Universal Robots PolyScope program: usb.urp

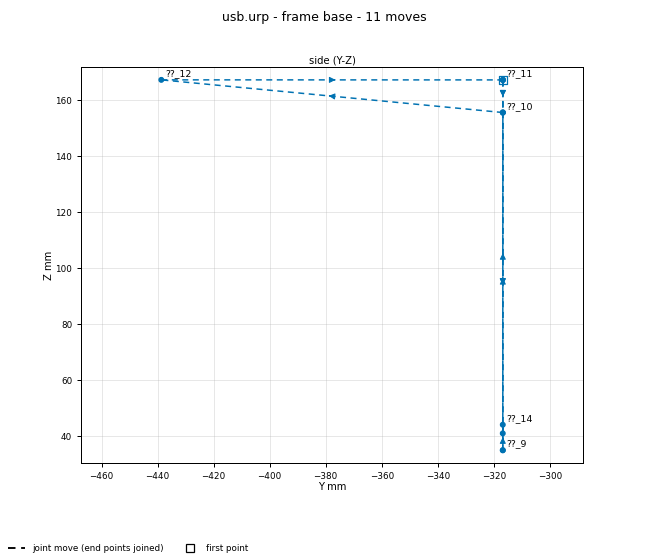
[picture p0: tool path of usb.urp in frame base, 11 of 11 moves have a stored position in this frame; points joined in program order, loops and branches not executed]
Program usb (installation=20240827 directory=/programs createdIn=5.15.1 lastSavedIn=5.15.1 robotSerialNumber=20245500285)
Calibrated DH parameters: a=[0.000097, -0.210459, -0.026602, 0.000137, 0.000078, 0]; d=[0.162601, 254.180657, -54.076236, -199.970743, 0.099615, 0.099684]; alpha=[1.569796, -0.001455, 0.001957, 1.570525, -1.571561, 0]; deltaTheta=[0, -1.053331, 8.839472, -1.50296, 0.000002, 0]
InitVariablesNode
Robot Program (runOnlyOnce=false)
  Script: usb = rpc_factory("xmlrpc","http://192.168.1.7:9120/RPC2")
  SuppressedNode
    MoveJ speed 60 deg/s, acceleration 80 deg/s^2 (useActiveTCP=true) feature=Base
      SuppressedNode
        Waypoint 路点_1: TCP in base x=280.909 y=-438.416 z=138.453 mm, rx=-0.0039 ry=2.6174 rz=0.002 rad; joints [90, -89.997, 120, -119.999, -60.002, 0] deg; TCP offset x=-0.17 y=0 z=192.95 mm, rx=0 ry=0 rz=0 rad
      Popup Message (haltProgram=false message=1 inputType=Text)
      Waypoint 路点_7: TCP in base x=280.9 y=-438.411 z=138.447 mm, rx=-0.0038 ry=3.1416 rz=0 rad; joints [107.671, -84.178, 107.406, -113.272, -90.026, 17.702] deg
      Waypoint 路点_2: TCP in base x=300.223 y=-316.781 z=157.956 mm, rx=0.0118 ry=-3.1414 rz=0.0001 rad; joints [115.532, -97.131, 117.117, -110.029, -90.021, 25.257] deg
      Waypoint 路点_3: TCP in base x=300.251 y=-316.773 z=100.612 mm, rx=0.0108 ry=-2.8383 rz=-0.0015 rad; joints [125.162, -84.56, 113.268, -108.499, -104.146, 36.158] deg
      Waypoint 路点_4: TCP in base x=300.243 y=-316.792 z=44.753 mm, rx=0.0106 ry=-2.8383 rz=-0.0015 rad; joints [125.158, -79.995, 117.672, -117.469, -104.165, 36.163] deg
      SuppressedNode
        Waypoint 路点_5: TCP in base x=301.229 y=-316.057 z=44.799 mm, rx=-0.0007 ry=-3.106 rz=-0.1207 rad; joints [115.546, -85.69, 123.783, -123.302, -89.838, 25.723] deg
      SuppressedNode
        Waypoint 路点_6: TCP in base x=280.91 y=-438.41 z=138.456 mm, rx=-0.0038 ry=2.6174 rz=0.002 rad; joints [89.999, -89.998, 120.001, -119.999, -60.001, 0.001] deg
      Waypoint ccc: TCP in base x=300.236 y=-316.791 z=40.853 mm, rx=0.0106 ry=-2.8383 rz=-0.0015 rad; joints [125.157, -79.629, 117.939, -118.1, -104.166, 36.162] deg
      Popup Message (haltProgram=false message=2 inputType=Text)
      Waypoint bbb: TCP in base x=300.214 y=-316.776 z=46.329 mm, rx=0.0105 ry=-3.1416 rz=-0.0001 rad; joints [115.525, -88.303, 127.676, -129.414, -90.051, 25.294] deg
      Waypoint aaa: TCP in base x=300.25 y=-316.768 z=32.092 mm, rx=0.0117 ry=-3.1415 rz=0.0001 rad; joints [115.535, -86.708, 128.728, -132.063, -90.063, 25.255] deg
  MoveJ speed 60 deg/s, acceleration 80 deg/s^2 (useActiveTCP=true) feature=Base
    Waypoint 路点_11: TCP in base x=302.488 y=-316.764 z=167.249 mm, rx=0.0098 ry=-3.1415 rz=0 rad; joints [115.808, -97.362, 115.876, -108.556, -90.01, 25.606] deg
    Script: usb.open()
    Popup Message (haltProgram=false message=1 inputType=Text)
    Waypoint 路点_10: TCP in base x=302.495 y=-316.788 z=155.612 mm, rx=0.0104 ry=-2.7358 rz=-0.0021 rad; joints [127.981, -84.22, 104.466, -95.426, -108.111, 40.089] deg
    Waypoint 路点_9: TCP in base x=302.521 y=-316.805 z=35.093 mm, rx=0.0103 ry=-2.7358 rz=-0.002 rad; joints [127.978, -75.737, 114.454, -113.902, -108.151, 40.091] deg
    Script: usb.close()
    Waypoint 路点_10: TCP in base x=302.495 y=-316.788 z=155.612 mm, rx=0.0104 ry=-2.7358 rz=-0.0021 rad; joints [127.981, -84.22, 104.466, -95.426, -108.111, 40.089] deg
    Popup Message (haltProgram=false message=1 inputType=Text)
  MoveJ speed 60 deg/s, acceleration 80 deg/s^2 (useActiveTCP=true) feature=Base
    Waypoint 路点_12: TCP in base x=302.499 y=-438.669 z=167.271 mm, rx=-0.0098 ry=3.1416 rz=0 rad; joints [109.96, -83.978, 102.672, -108.739, -90.019, 19.776] deg
    Popup Message (haltProgram=false message=1 inputType=Text)
    SuppressedNode
      Script: usb.open()
    SuppressedNode
      Popup Message (haltProgram=false message=1 inputType=Text)
    SuppressedNode
      Script: usb.close()
    SuppressedNode
      Popup Message (haltProgram=false message=1 inputType=Text)
    Waypoint 路点_11: TCP in base x=302.488 y=-316.764 z=167.249 mm, rx=0.0098 ry=-3.1415 rz=0 rad; joints [115.808, -97.362, 115.876, -108.556, -90.01, 25.606] deg
    Waypoint 路点_10: TCP in base x=302.495 y=-316.788 z=155.612 mm, rx=0.0104 ry=-2.7358 rz=-0.0021 rad; joints [127.981, -84.22, 104.466, -95.426, -108.111, 40.089] deg
    SuppressedNode
      Waypoint 路点_14: TCP in base x=302.527 y=-316.813 z=44.199 mm, rx=0.0104 ry=-2.7358 rz=-0.0019 rad; joints [127.98, -76.564, 113.866, -112.489, -108.15, 40.091] deg
    SuppressedNode
      Popup Message (haltProgram=false message=1 inputType=Text)
    Waypoint 路点_9: TCP in base x=302.521 y=-316.805 z=35.093 mm, rx=0.0103 ry=-2.7358 rz=-0.002 rad; joints [127.978, -75.737, 114.454, -113.902, -108.151, 40.091] deg
    Wait Sleep waitTime=0.1
    Script: usb.open()
    SuppressedNode
      Popup Message (haltProgram=false message=1 inputType=Text)
    Waypoint 路点_14: TCP in base x=302.527 y=-316.813 z=44.199 mm, rx=0.0104 ry=-2.7358 rz=-0.0019 rad; joints [127.98, -76.564, 113.866, -112.489, -108.15, 40.091] deg
    Script: usb.close()
    SuppressedNode
      Popup Message (haltProgram=false message=1 inputType=Text)
    Waypoint 路点_13: TCP in base x=302.53 y=-316.817 z=41.115 mm, rx=0.0104 ry=-2.7358 rz=-0.0019 rad; joints [127.98, -76.288, 114.069, -112.97, -108.151, 40.089] deg
    Script: usb.open()
    Waypoint 路点_11: TCP in base x=302.488 y=-316.764 z=167.249 mm, rx=0.0098 ry=-3.1415 rz=0 rad; joints [115.808, -97.362, 115.876, -108.556, -90.01, 25.606] deg
